FUNCTION_BLOCK AxisControlLogic
VAR_IN_OUT //pass by reference
	control					:CTR_SIGNALS_INTERNAL;
END_VAR
VAR
	couple					:BOOL	:= 0;
	revCouple				:BOOL	:= 0;
	prevCoupleControl		:BOOL	:= 0;
	prevRevCouple			:BOOL	:= 0;
END_VAR

IF GVL_MOTION.EXT_CTR.AxesEn AND NOT Main.eStop THEN
	control.Enable 						:= TRUE;
	control.CouplePowerEn  				:= TRUE;
ELSE
	control.Enable						:= FALSE;
	control.CouplePowerEn 				:= FALSE;
END_IF


//axis coupling control
//toggle flip flop for state change on each rising edge transition
IF control.CoupleControl THEN
	//cant set coupling axis inside program/function block. assignments in MAIN
	control.CoupleControl				:= FALSE;
	CASE control.CoupleState OF
		0:
			control.ExecuteUncouple  	:= FALSE;
			control.ExecuteCouple 		:= TRUE;
			control.CoupleState 		:= 1;
		1:
			control.ExecuteCouple 		:= FALSE;
			control.ExecuteUncouple 	:= TRUE;	
			control.CoupleState 		:= 0;
	END_CASE
END_IF

//prevCoupleControl 						:= control.CoupleControl;

END_FUNCTION_BLOCK

(* stored: Version 1.1.0.1, ProductVersion 3.1.4026.12
   POU AxisControlLogic: Id {5a657959-1248-4dfd-a9b9-189be3061d05}, SpecialFunc None *)
